// TIA Portal V20 export
TYPE "LER_typeUnitHmiData"
// stored: Access Published
   STRUCT
      PartType : Byte;   // Normal model: 1 -50Master gauge.1: 51Master gauge.2: 52Master gauge.3: 53reserved: 54-98Dry run/Idle: 99 (run without part)
      PartStatus : Byte;   // 0: wrong data1: No part2: OK part3: NOK part4: gauge part5: inspection part6: sampled part7-: reserved
   END_STRUCT;
END_TYPE
